{attribute addProperty BoxType "EK1960-0000-0021"}
{attribute addProperty Id "FSoE_InputsFSoE_Inputs_91F6EA7112015FSoE_OutputsFSoE_Outputs_DB0FA8F712015"}
{attribute addProperty CRC "3657549630"}
{attribute addProperty SizeInBites "240"}
{attribute addProperty SizeInBytes "30"}
TYPE Module_1_FSoE_DA01C73E :
STRUCT
	{attribute addProperty Name "FSoE_Inputs"}
	FSoE_Inputs  : FSoE_Inputs_91F6EA71;
	{attribute addProperty Name "FSoE_Outputs"}
	FSoE_Outputs  : FSoE_Outputs_DB0FA8F7;
END_STRUCT
END_TYPE

(* stored: Version 1.2.0.0, ProductVersion 3.1.4024.9
   DUT Module_1_FSoE_DA01C73E: Id {60b3e9ab-2dfd-4866-99cc-1f709c8ce61a} *)
